(* IEC 61131-3 sources: Lasal/CPU_5344_V01/Class/stopSafetyAndOpenDoor, 1 file *)

(* ---- stopSafetyAndOpenDoor.st ---- *)
(*!
<Class
	Name               = "stopSafetyAndOpenDoor"
	Revision           = "0.0"
	RealtimeTask       = "false"
	CyclicTask         = "true"
	DefCyclictime      = "10 ms"
	BackgroundTask     = "false"
	Sigmatek           = "false"
	OSInterface        = "false"
	HighPriority       = "false"
	Automatic          = "false"
	UpdateMode         = "Prescan"
	SharedCommandTable = "true"
	Objectsize         = "(284,120)">
	<Channels>
		<Server Name="ClassSvr" Visualized="false" Initialize="false" WriteProtected="true" Retentive="false"/>
		<Server Name="openSawDoor" Visualized="true" Initialize="false" WriteProtected="false" Retentive="false"/>
		<Server Name="readOpenSawDoor" Visualized="false" Initialize="false" WriteProtected="true" Retentive="false"/>
		<Server Name="resetSafety" Visualized="false" Initialize="false" WriteProtected="true" Retentive="false"/>
		<Server Name="sparMaxButtonTime" Visualized="false" Initialize="true" DefValue="240000" WriteProtected="false" Retentive="File"/>
		<Server Name="stopSafety" Visualized="false" Initialize="false" WriteProtected="true" Retentive="false"/>
		<Client Name="iPBresetSafety" Required="true" Internal="false"/>
		<Client Name="iSafetyState" Required="true" Internal="false"/>
		<Client Name="iStopSafetyAllowed" Required="true" Internal="false"/>
	</Channels>
</Class>
*)
stopSafetyAndOpenDoor : CLASS
  //Servers:
	ClassSvr 	: SvrChCmd_DINT;
	resetSafety 	: SvrCh_DINT;
	openSawDoor 	: SvrCh_DINT;
	stopSafety 	: SvrCh_DINT;
	sparMaxButtonTime 	: SvrCh_UDINT;
	readOpenSawDoor 	: SvrCh_DINT;
  //Clients:
	iPBresetSafety 	: CltCh_DINT;
	iStopSafetyAllowed 	: CltCh_DINT;
	iSafetyState 	: CltCh_DINT;
  //Variables:
		tmpButtonTime 	: UDINT;
		oldPBresetSafety 	: DINT;
  //Functions:

	FUNCTION VIRTUAL GLOBAL CyWork
		VAR_INPUT
			EAX 	: UDINT;
		END_VAR
		VAR_OUTPUT
			state (EAX) 	: UDINT := READY;
		END_VAR;

	FUNCTION VIRTUAL GLOBAL openSawDoor::Write
		VAR_INPUT
			input (EAX) 	: DINT;
		END_VAR
		VAR_OUTPUT
			result (EAX) 	: DINT;
		END_VAR;

	FUNCTION VIRTUAL GLOBAL readOpenSawDoor::Read
		VAR_OUTPUT
			output (EAX) 	: DINT;
		END_VAR;
  //Tables:
	FUNCTION @STD
		VAR_OUTPUT
			ret_code	: CONFSTATES;
		END_VAR;
	FUNCTION GLOBAL TAB @CT_;
END_CLASS;

FUNCTION VIRTUAL GLOBAL stopSafetyAndOpenDoor::CyWork
	VAR_INPUT
		EAX 	: UDINT;
	END_VAR
	VAR_OUTPUT
		state (EAX) 	: UDINT;(* := READY *)
	END_VAR

  iPBresetSafety := iPBresetSafety.Read();
  iStopSafetyAllowed := iStopSafetyAllowed.Read();
  iSafetyState:= iSafetyState.Read();

  IF iPBresetSafety & iStopSafetyAllowed & oldPBresetSafety=0 THEN
    StopSafety:= 0; //means stop it
  END_IF;
  IF iStopSafetyAllowed=0 | iSafetyState=0 THEN
    StopSafety:= 1; //means just go on
  END_IF;

  IF stopSafety= 1 THEN
    resetSafety:= iPBresetSafety;
  END_IF;

  IF iSafetyState= 1 | (ops.tAbsolute-tmpButtonTime> sparMaxButtonTime) THEN
    openSawDoor:= 0; //in screen this one can be enabled for one minute
  END_IF;

  oldPBresetSafety:= iPBresetSafety;

END_FUNCTION

FUNCTION VIRTUAL GLOBAL stopSafetyAndOpenDoor::openSawDoor::Write
	VAR_INPUT
		input (EAX) 	: DINT;
	END_VAR
	VAR_OUTPUT
		result (EAX) 	: DINT;
	END_VAR

  IF iSafetyState= 0 THEN
    openSawDoor := input;
    tmpButtonTime:= ops.tAbsolute;
  END_IF;
	result := openSawDoor;

END_FUNCTION

FUNCTION VIRTUAL GLOBAL stopSafetyAndOpenDoor::readOpenSawDoor::Read
	VAR_OUTPUT
		output (EAX) 	: DINT;
	END_VAR

  readOpenSawDoor:= openSawDoor;
	output := readOpenSawDoor;

END_FUNCTION
